{attribute 'qualified_only'}
{attribute 'strict'}
TYPE E_GeneralStatus :
(
	NONE := 0,
	STOP,
	BUSY,
	DONE,
	ERROR,
	INPUT_ERROR,
	INTERRUPT
);
END_TYPE

(* stored: Version 1.1.0.1, ProductVersion 3.1.4024.11
   EnumerationTextList E_GeneralStatus: Id {c9ac1dff-20af-4621-8bbb-e71ea610e75d} *)
